{attribute 'linkalways'} 
{attribute 'no_explicit_call' := 'This FB is a CLASS and must be accessed using methods or properties'}
{attribute 'enable_dynamic_creation'}
FUNCTION_BLOCK _ETcVnDataLayout EXTENDS EnumDatatypeBase
VAR
	localData : ETcVnDataLayout;
	activeData : REFERENCE TO ETcVnDataLayout;
	enumBaseDatatype : _ULINT(localData);
END_VAR

METHOD PRIVATE AddLocalEnumeration
VAR_INPUT
	Enumeration : T_MAXSTRING;
	Value : ETcVnDataLayout;
END_VAR
AddEnumeration(Enumeration, Value);
END_METHOD

PROPERTY PUBLIC Address : PVOID
GET
Address := ADR(activeData);
END_GET
END_PROPERTY

METHOD PUBLIC ClearReference
VAR_INPUT
END_VAR
activeData REF= localData;
SetBaseDatatypeReference();
END_METHOD

METHOD PUBLIC Clone : I_Datatype
VAR
    pClone : POINTER TO _ETcVnDataLayout;
END_VAR
pClone := __NEW(_ETcVnDataLayout(InitialValue := Value));
Clone := pClone^;
END_METHOD

METHOD FB_init : BOOL
VAR_INPUT
	bInitRetains : BOOL; // if TRUE, the retain variables are initialized (warm start / cold start)
	bInCopyCode : BOOL;  // if TRUE, the instance afterwards gets moved into the copy code (online change)
	InitialValue : ETcVnDataLayout;
END_VAR
localData := InitialValue;
AddBaseDatatype(enumBaseDatatype);
ClearReference();

AddLocalEnumeration('TCVN_DL_DEFAULT', ETcVnDataLayout.TCVN_DL_DEFAULT);
AddLocalEnumeration('TCVN_DL_2D_HW', ETcVnDataLayout.TCVN_DL_2D_HW);
AddLocalEnumeration('TCVN_DL_2D_WH', ETcVnDataLayout.TCVN_DL_2D_WH);
AddLocalEnumeration('TCVN_DL_3D_CHW', ETcVnDataLayout.TCVN_DL_3D_CHW);
AddLocalEnumeration('TCVN_DL_3D_HWC', ETcVnDataLayout.TCVN_DL_3D_HWC);
AddLocalEnumeration('TCVN_DL_4D_NCHW', ETcVnDataLayout.TCVN_DL_4D_NCHW);
AddLocalEnumeration('TCVN_DL_4D_NHWC', ETcVnDataLayout.TCVN_DL_4D_NHWC);
END_METHOD

PROPERTY PUBLIC Identifier : T_MAXSTRING
GET
Identifier := 'ETcVnDataLayout';
END_GET
END_PROPERTY

METHOD IsEnumeratorValueEqual : BOOL
VAR_INPUT
	Enumerator : I_KeyValueForwardEnumerator;
END_VAR
VAR
	storedValue : ETcVnDataLayout;
END_VAR
IF NOT Enumerator.TryGet(storedValue) THEN
	RETURN;
END_IF

IsEnumeratorValueEqual := storedValue = activeData;
END_METHOD

METHOD PUBLIC MakeReferenceTo
VAR_INPUT
	ReferenceTarget : REFERENCE TO ETcVnDataLayout;
END_VAR
activeData REF= ReferenceTarget;
SetBaseDatatypeReference();
END_METHOD

METHOD PROTECTED SetBaseDatatypeReference
VAR_INPUT
END_VAR
enumBaseDatatype.MakeReferenceTo(activeData);
END_METHOD

PROPERTY PUBLIC Size : UDINT
GET
Size := SIZEOF(activeData);
END_GET
END_PROPERTY

METHOD TryMakeReferenceTo : BOOL
VAR_INPUT
	Target : I_Datatype;
END_VAR
VAR
	pTargetData : POINTER TO ETcVnDataLayout;
END_VAR
IF NOT IsEquivalentTo(Target) THEN
	RETURN;
END_IF

pTargetData := Target.Address;
activeData REF= pTargetData^;
SetBaseDatatypeReference();
TryMakeReferenceTo := TRUE;
END_METHOD

PROPERTY PUBLIC Value : ETcVnDataLayout
GET
Value := activeData;
END_GET
SET
activeData := Value;
END_SET
END_PROPERTY

END_FUNCTION_BLOCK

(* stored: Version 1.1.0.1, ProductVersion 3.1.4024.15
   POU _ETcVnDataLayout: Id {b3d4ed9b-a7c8-0713-3cca-f81c1ff7ab7f}, SpecialFunc None
   Folder Core: Id {6cc8a929-8519-0d5f-2cae-29debf45c801}
   Folder Protected: Id {e7e5c463-b947-049b-3d20-840f3d3c5db6}
   Folder Customize: Id {a07d372b-31ff-02f6-27d5-e9f590abb31f}
   Folder Constructor: Id {414c6788-9e33-0bbe-0abb-9da33a72b177}
   Folder Private: Id {6df5d032-31d5-0d58-04b7-cce0a7eafa10}
   Folder Protected: Id {24abdaa0-2f52-04cd-24d9-9c60ce719747}
   Method AddLocalEnumeration: Id {7fba1930-db76-08e9-3b2e-3aa8db2f96e9}
   Property Address: Id {afbdadc3-1476-022c-0c21-a3534090bb93}
   Get Get: Id {cca86d51-4728-0f7e-16f1-b58b6dea8284}
   Method ClearReference: Id {c1afc26f-1036-0e22-34eb-5ac67a1cd69f}
   Method Clone: Id {89616688-0dfb-02ec-30ae-4c2f8e9f1144}
   Method FB_init: Id {438ff0a8-c439-046c-0dea-0df768ca7cdc}
   Property Identifier: Id {c4a6bd90-a0ec-0dae-0e00-4c4b6bd61e74}
   Get Get: Id {1e7cd755-43b6-0673-2a2c-d688cc58270d}
   Method IsEnumeratorValueEqual: Id {7f7108bc-1463-0a49-1a38-eec01490ff8b}
   Method MakeReferenceTo: Id {846206ad-115c-0ade-3368-0c3f79de794e}
   Method SetBaseDatatypeReference: Id {f19d8e72-aed0-0f8b-2c83-6329bfc18cf8}
   Property Size: Id {0a70cea4-3d93-03c1-0feb-44cc9f00a402}
   Get Get: Id {22ddbc75-14cb-08d9-1ef3-e7e1884b417b}
   Method TryMakeReferenceTo: Id {04f0e290-ba84-01c8-2df3-e8c4f44b6acb}
   Property Value: Id {dc0d6b69-e6fb-0470-0f7e-623a20d3452a}
   Get Get: Id {f4072b0b-96c0-006b-3b07-8066887ce5c7}
   Set Set: Id {02f4a883-5ea8-02ca-0f10-207db8fad3e3} *)
